// SIMATIC STEP 7 (V5.x) project Platform_V1_5
// CPU: CPU 312IFM
// CPU: CPU 313
// station: Hardware
// station: Slave
// station: P_ADR_BUS
// station: P_ADR_BUS
// station: Configuration
// station: Hardware
// station: Master
// station: P_ADR_BUS
// program: S7 Program(1)
// program: S7 Program(3)

SYMBOL_TABLE
"Ingangen.Doorsturen"	FC 1	FC 1
"Watchdog"	FC 2	FC 2
"Uitgangen.Prioriteit"	FC 3	FC 3
"Start"	I 0.0	BOOL
"Stop"	I 0.1	BOOL
"Piston A in"	I 0.2	BOOL
"Piston A uit"	I 0.3	BOOL
"Piston A onder"	I 0.4	BOOL
"Piston A boven"	I 0.5	BOOL
"Piston B in"	I 0.6	BOOL
"Piston B uit"	I 0.7	BOOL
"Piston B onder"	I 124.0	BOOL
"Piston B boven"	I 124.1	BOOL
"Proxi Pos 1"	I 124.2	BOOL
"Proxi Pos 2"	I 124.3	BOOL
"Watch.Slave.Master.Go"	M 4.0	BOOL	// Van slave Naar Master
"Watch.Slave.Master.Back"	M 4.1	BOOL	// Van slave Naar master
"Watch.Master.Slave.Go"	M 4.2	BOOL
"Watch.Master.Slave.Back"	M 4.3	BOOL
"Watch.Slave.Sim.Go"	M 4.4	BOOL
"Watch.Slave.Sim.back"	M 4.5	BOOL
"Levens.Bit"	M 10.0	BOOL
"Levens.Bit.Fout"	M 10.1	BOOL
"Ingangen 0.x"	MB 0	BYTE
"Ingangen 124.x"	MB 1	BYTE
"Uitgangen 0.x"	MB 2	BYTE
"Uitgangen 124.x"	MB 3	BYTE
"Motor Rechts"	Q 0.1	BOOL
"Piston A Op-Neer"	Q 0.2	BOOL
"Piston A Uit-In"	Q 0.3	BOOL
"Piston B Op-Neer"	Q 0.4	BOOL
"Piston B Uit-In"	Q 0.5	BOOL
"Sign.Rood"	Q 0.6	BOOL
"Motor Links"	Q 124.0	BOOL
"Extend.proxi2"	T 0	TIMER
"Levens.bit.1"	T 1	TIMER
"Levens.bit.2"	T 2	TIMER
END_SYMBOL_TABLE

FUNCTION "Ingangen.Doorsturen" : VOID	// FC 1
VERSION : 0.1
BEGIN
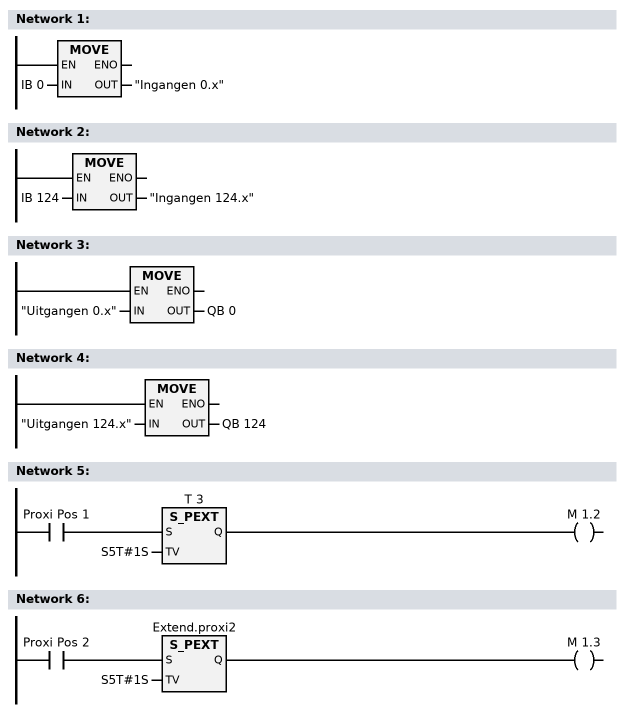
NETWORK
TITLE =
      L     IB 0;
      T     "Ingangen 0.x";
      NOP   0;
NETWORK
TITLE =
      L     IB 124;
      T     "Ingangen 124.x";
      NOP   0;
NETWORK
TITLE =
      L     "Uitgangen 0.x";
      T     QB 0;
      NOP   0;
NETWORK
TITLE =
      L     "Uitgangen 124.x";
      T     QB 124;
      NOP   0;
NETWORK
TITLE =
      A     "Proxi Pos 1";
      L     S5T#1S;
      SE    T 3;
      NOP   0;
      NOP   0;
      NOP   0;
      A     T 3;
      =     M 1.2;
NETWORK
TITLE =
      A     "Proxi Pos 2";
      L     S5T#1S;
      SE    "Extend.proxi2";
      NOP   0;
      NOP   0;
      NOP   0;
      A     "Extend.proxi2";
      =     M 1.3;
END_FUNCTION

FUNCTION "Watchdog" : VOID	// FC 2
VERSION : 0.1
BEGIN
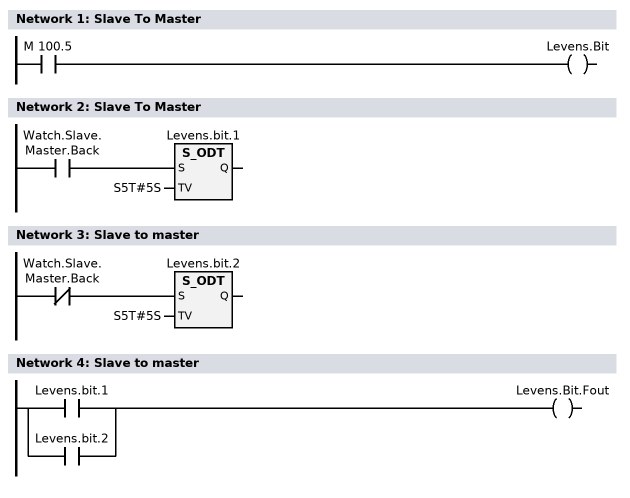
NETWORK
TITLE = Slave To Master
      A     M 100.5;
      =     "Levens.Bit";
NETWORK
TITLE = Slave To Master
      A     "Watch.Slave.Master.Back";
      L     S5T#5S;
      SD    "Levens.bit.1";
      NOP   0;
      NOP   0;
      NOP   0;
      NOP   0;
NETWORK
TITLE = Slave to master
      AN    "Watch.Slave.Master.Back";
      L     S5T#5S;
      SD    "Levens.bit.2";
      NOP   0;
      NOP   0;
      NOP   0;
      NOP   0;
NETWORK
TITLE = Slave to master
      O     "Levens.bit.1";
      O     "Levens.bit.2";
      =     "Levens.Bit.Fout";
END_FUNCTION

FUNCTION "Uitgangen.Prioriteit" : VOID	// FC 3
VERSION : 0.1
BEGIN
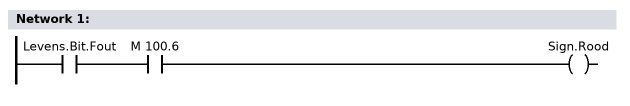
NETWORK
TITLE =
      A     "Levens.Bit.Fout";
      A     M 100.6;
      =     "Sign.Rood";
END_FUNCTION

ORGANIZATION_BLOCK OB 1
TITLE = "Main Program Sweep (Cycle)"
VERSION : 0.1
VAR_TEMP
  OB1_EV_CLASS : BYTE ;	//Bits 0-3 = 1 (Coming event), Bits 4-7 = 1 (Event class 1)
  OB1_SCAN_1 : BYTE ;	//1 (Cold restart scan 1 of OB 1), 3 (Scan 2-n of OB 1)
  OB1_PRIORITY : BYTE ;	//Priority of OB Execution
  OB1_OB_NUMBR : BYTE ;	//1 (Organization block 1, OB1)
  OB1_RESERVED_1 : BYTE ;	//Reserved for system
  OB1_RESERVED_2 : BYTE ;	//Reserved for system
  OB1_PREV_CYCLE : INT ;	//Cycle time of previous OB1 scan (milliseconds)
  OB1_MIN_CYCLE : INT ;	//Minimum cycle time of OB1 (milliseconds)
  OB1_MAX_CYCLE : INT ;	//Maximum cycle time of OB1 (milliseconds)
  OB1_DATE_TIME : DATE_AND_TIME ;	//Date and time OB1 started
END_VAR
BEGIN
NETWORK
TITLE =
      CALL  "Ingangen.Doorsturen";
      CALL  "Watchdog";
      CALL  "Uitgangen.Prioriteit";
END_ORGANIZATION_BLOCK

// (several symbol tables fit these blocks; global names not applied)

FUNCTION FC 1 : VOID
VERSION : 0.1
BEGIN
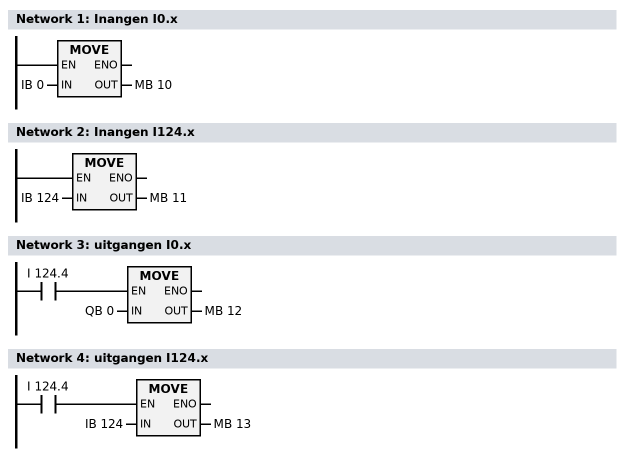
NETWORK
TITLE = Inangen I0.x
      L     IB 0;
      T     MB 10;
      NOP   0;
NETWORK
TITLE = Inangen I124.x
      L     IB 124;
      T     MB 11;
      NOP   0;
NETWORK
TITLE = uitgangen I0.x
      A     I 124.4;
      JNB   _001;
      L     QB 0;
      T     MB 12;
_001: NOP   0;
NETWORK
TITLE = uitgangen I124.x
      A     I 124.4;
      JNB   _002;
      L     IB 124;
      T     MB 13;
_002: NOP   0;
END_FUNCTION

ORGANIZATION_BLOCK OB 1
TITLE = "Main Program Sweep (Cycle)"
VERSION : 0.1
VAR_TEMP
  OB1_EV_CLASS : BYTE ;	//Bits 0-3 = 1 (Coming event), Bits 4-7 = 1 (Event class 1)
  OB1_SCAN_1 : BYTE ;	//1 (Cold restart scan 1 of OB 1), 3 (Scan 2-n of OB 1)
  OB1_PRIORITY : BYTE ;	//Priority of OB Execution
  OB1_OB_NUMBR : BYTE ;	//1 (Organization block 1, OB1)
  OB1_RESERVED_1 : BYTE ;	//Reserved for system
  OB1_RESERVED_2 : BYTE ;	//Reserved for system
  OB1_PREV_CYCLE : INT ;	//Cycle time of previous OB1 scan (milliseconds)
  OB1_MIN_CYCLE : INT ;	//Minimum cycle time of OB1 (milliseconds)
  OB1_MAX_CYCLE : INT ;	//Maximum cycle time of OB1 (milliseconds)
  OB1_DATE_TIME : DATE_AND_TIME ;	//Date and time OB1 started
END_VAR
BEGIN
// (block stored without names or comments; labels and parameter names are numbered)
END_ORGANIZATION_BLOCK

SYMBOL_TABLE
"Productie_teller_Station"	C 0	COUNTER
"Productie_teller_Stat_A"	C 1	COUNTER
"Productie_teller_Stat_B"	C 2	COUNTER
"Productie_teller_In_Waar"	C 3	COUNTER
"SIM.Positie.Staven"	C 4	COUNTER
"SIM.OB1"	DB 2	DB 2	// Simualtie
"SIM.USERS"	DB 3	DB 3
"Positionering"	DB 4	DB 4
"Uitgangen Sturen"	FC 1	FC 1
"Timers + Counters"	FC 2	FC 2
"Grafcet Station A"	FC 3	FC 3
"Grafcet Station B"	FC 4	FC 4
"Simulatie_Run"	FC 5	FC 5
"Opstart_FC"	FC 6	FC 6
"Grafcet_Platform"	FC 7	FC 7	// Grafcet_Platform
"Ingang -> Merker"	FC 8	FC 8
"DB_Function"	FC 9	FC 9
"SIM.OB100"	FC 10	FC 10
"SIM.user"	FC 11	FC 11
"Positionering_balken"	FC 12	FC 12
"Sub_routine"	FC 14	FC 14
"Opstart_subroutine"	FC 15	FC 15
"Sub_routine_gelijk"	FC 16	FC 16
"Sub_route_Station_samen"	FC 17	FC 17
"SIM.SUBR.Y-As"	FC 19	FC 19
"SIM.LOGIN"	FC 20	FC 20
"SIM.Move.X-As"	FC 21	FC 21
"SIM.BALK.Reset"	FC 22	FC 22
"Stap 0.0"	M 0.0	BOOL
"Stap 0.1"	M 0.1	BOOL
"Stap 0.2"	M 0.2	BOOL
"Stap 0.3"	M 0.3	BOOL
"Stap 0.4"	M 0.4	BOOL
"Stap 0.5"	M 0.5	BOOL
"Stap 1.1"	M 1.1	BOOL
"Stap 1.2"	M 1.2	BOOL
"Stap 1.3"	M 1.3	BOOL
"Stap 1.4"	M 1.4	BOOL
"Stap 1.5"	M 1.5	BOOL
"Stap 2.0"	M 2.0	BOOL
"Stap 2.1"	M 2.1	BOOL
"Stap 2.2"	M 2.2	BOOL
"Stap 2.3"	M 2.3	BOOL
"Stap 2.4"	M 2.4	BOOL
"Stap 2.5"	M 2.5	BOOL
"Start"	M 5.0	BOOL
"Stop"	M 5.1	BOOL
"Piston A in"	M 5.2	BOOL
"Piston A uit"	M 5.3	BOOL
"Piston A onder"	M 5.4	BOOL
"Piston A boven"	M 5.5	BOOL
"Piston B in"	M 5.6	BOOL
"Piston B uit"	M 5.7	BOOL
"Piston B onder"	M 6.0	BOOL
"Piston B boven"	M 6.1	BOOL
"Proxi Pos 1"	M 6.2	BOOL
"Proxi Pos 2"	M 6.3	BOOL
"Motor Rechts"	M 7.1	BOOL
"Piston A Op-Neer"	M 7.2	BOOL
"Piston A Uit-In"	M 7.3	BOOL
"Piston B Op-Neer"	M 7.4	BOOL
"Piston B Uit-In"	M 7.5	BOOL
"Sign.Rood"	M 7.6	BOOL
"Sign.Groen"	M 7.7	BOOL
"Motor Links"	M 8.0	BOOL
"Opstart"	M 10.0	BOOL
"SIM.reset.C4"	M 10.1	BOOL
"P.M10.2"	M 10.2	BOOL
"SIM.opstart.5S"	M 10.3	BOOL
"admin"	M 11.0	BOOL
"monitor"	M 11.1	BOOL
"operate"	M 11.2	BOOL
"user"	M 11.3	BOOL
"SIM.User.Login"	M 11.4	BOOL
"SIM.User.logout"	M 11.5	BOOL
"SIM.USER.ERROR"	M 11.6	BOOL
"Sim.Start.Postitionering"	M 24.0	BOOL
"Postitionering.Station.A"	M 24.1	BOOL
"Postitionering.Station.B"	M 24.2	BOOL
"Postitionering.Return"	M 24.3	BOOL
"SIM.Positie.Save"	M 24.4	BOOL
"SIM.Positie.Zoom"	M 24.5	BOOL
"Balk1"	M 25.0	BOOL
"Blak2"	M 25.1	BOOL
"Balk3"	M 25.2	BOOL
"Balk4"	M 25.3	BOOL
"Balk5"	M 25.4	BOOL
"Balk6"	M 25.5	BOOL
"Balk7"	M 25.6	BOOL
"Balk8"	M 25.7	BOOL
"Test Piston A"	M 30.0	BOOL
"Fout Controle station A"	M 30.1	BOOL
"Fout Reset station A"	M 30.2	BOOL
"Test station B"	M 30.3	BOOL
"Fout Controle station B"	M 30.4	BOOL
"Fout_Motor"	M 30.5	BOOL
"Foint Station_A_B"	M 30.6	BOOL
"Stop Meker"	M 30.7	BOOL
"DBW0 == DBW2"	M 31.0	BOOL
"DBW0 < DBW2"	M 31.1	BOOL
"DBW0 != 0"	M 31.2	BOOL
"SIM.Start.StaA"	M 31.3	BOOL
"SIM.Start.StaB"	M 31.4	BOOL
"SIM.Start"	M 31.5	BOOL
"SIM.Stop"	M 31.6	BOOL
"DBW0 == 0"	M 32.0	BOOL
"INI.Stations"	M 33.0	BOOL
"Start Stat A + B"	M 33.1	BOOL
"Blinker 5s"	M 100.5	BOOL
"Restart"	M 101.1	BOOL
"Ingangen 0.x"	MB 5	BYTE
"Ingangen 124.x"	MB 6	BYTE
"Uitgangen 0.x"	MB 7	BYTE
"Uitgangen 124.x"	MB 8	BYTE
"Positie.balken"	MB 25	BYTE
"SIM.C.Positie.BCD"	MW 12	WORD	// Balk die zich bevind voor de sensoren(bcd waarde)
"SIM.C.Positie.INT"	MW 14	INT	// Balk die zich bevind voor de sensoren(int waarde)
"SIM.C.Postie.Stat.A"	MW 16	INT	// Balk die zich bevind voor station A
"SIM.C.Postie.Stat.B"	MW 18	INT	// Balk due zich bevind voor station B
"SIM.Station.A"	MW 20	WORD
"SIM.Station.B"	MW 22	WORD
"COMPLETE RESTART"	OB 100	OB 100	// Complete Restart
"Motor controler"	T 0	TIMER
"Timer Contr Neer A"	T 1	TIMER
"Timer contr uit A"	T 2	TIMER
"Timer contr uit B"	T 3	TIMER
"Timer contr neer B"	T 4	TIMER
"Hori Station B"	T 5	TIMER
"Verti Station B"	T 6	TIMER
"SIM.SUBR.T1"	T 7	TIMER
"SIM.SUBR.T2"	T 8	TIMER
"SIM.User.Error.T"	T 9	TIMER
"Vertraging.Station.off"	T 10	TIMER
"Vertraging.Station.Aan"	T 11	TIMER
END_SYMBOL_TABLE

FUNCTION "Uitgangen Sturen" : VOID	// FC 1
VERSION : 0.1
BEGIN
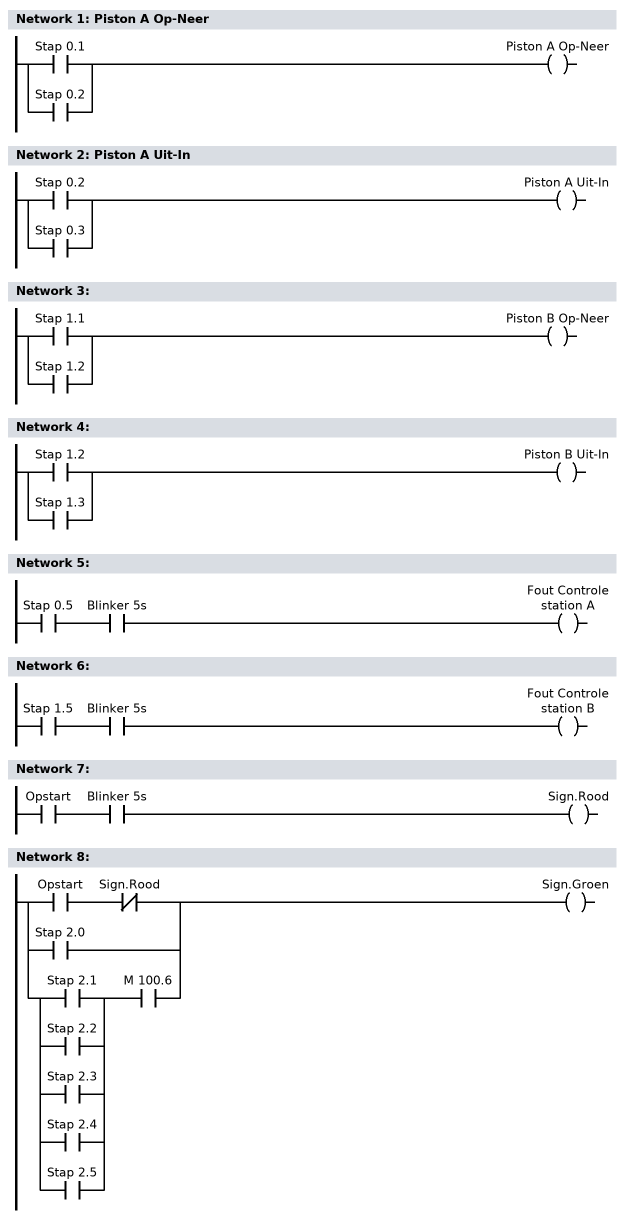
NETWORK
TITLE = Piston A Op-Neer
      O     "Stap 0.1";
      O     "Stap 0.2";
      =     "Piston A Op-Neer";
NETWORK
TITLE = Piston A Uit-In
      O     "Stap 0.2";
      O     "Stap 0.3";
      =     "Piston A Uit-In";
NETWORK
TITLE =
      O     "Stap 1.1";
      O     "Stap 1.2";
      =     "Piston B Op-Neer";
NETWORK
TITLE =
      O     "Stap 1.2";
      O     "Stap 1.3";
      =     "Piston B Uit-In";
NETWORK
TITLE =
      A     "Stap 0.5";
      A     "Blinker 5s";
      =     "Fout Controle station A";
NETWORK
TITLE =
      A     "Stap 1.5";
      A     "Blinker 5s";
      =     "Fout Controle station B";
NETWORK
TITLE =
      A     "Opstart";
      A     "Blinker 5s";
      =     "Sign.Rood";
NETWORK
TITLE =
      A     "Opstart";
      AN    "Sign.Rood";
      O     "Stap 2.0";
      O;
      A(;
      O     "Stap 2.1";
      O     "Stap 2.2";
      O     "Stap 2.3";
      O     "Stap 2.4";
      O     "Stap 2.5";
      );
      A     M 100.6;
      =     "Sign.Groen";
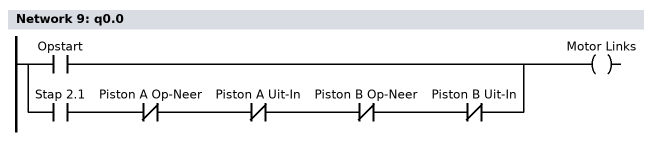
NETWORK
TITLE = q0.0
      O     "Opstart";
      O;
      A     "Stap 2.1";
      AN    "Piston A Op-Neer";
      AN    "Piston A Uit-In";
      AN    "Piston B Op-Neer";
      AN    "Piston B Uit-In";
      =     "Motor Links";
END_FUNCTION

FUNCTION "Timers + Counters" : VOID	// FC 2
VERSION : 0.1
BEGIN
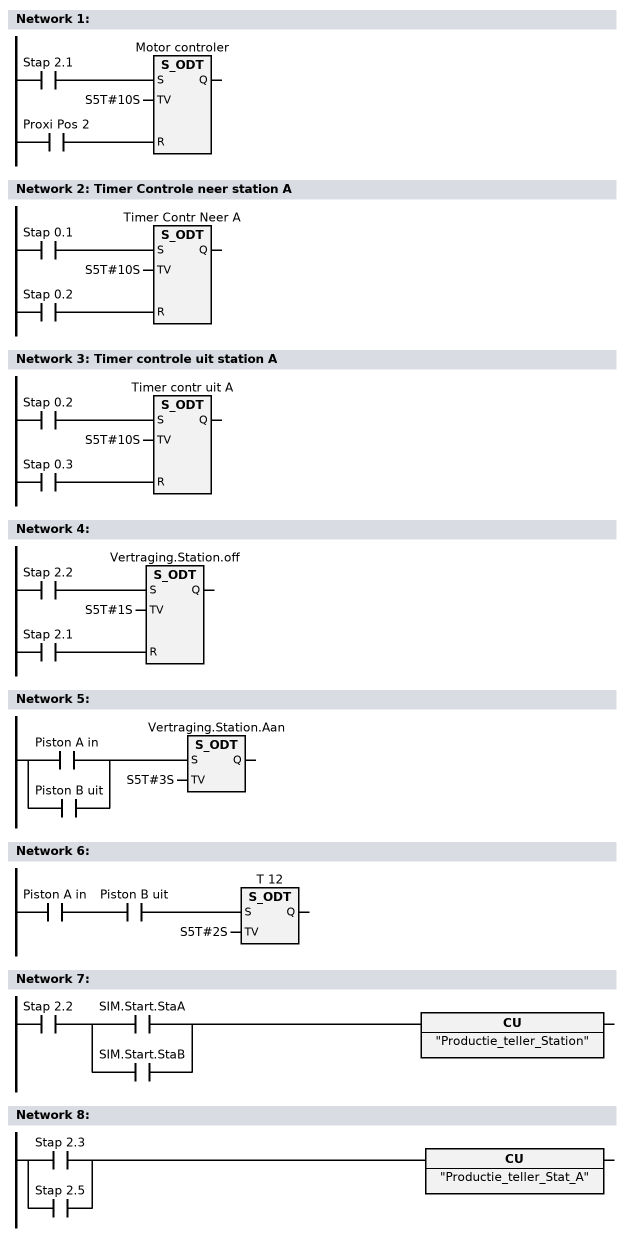
NETWORK
TITLE =
      A     "Stap 2.1";
      L     S5T#10S;
      SD    "Motor controler";
      A     "Proxi Pos 2";
      R     "Motor controler";
      NOP   0;
      NOP   0;
      NOP   0;
NETWORK
TITLE = Timer Controle neer station A
      A     "Stap 0.1";
      L     S5T#10S;
      SD    "Timer Contr Neer A";
      A     "Stap 0.2";
      R     "Timer Contr Neer A";
      NOP   0;
      NOP   0;
      NOP   0;
NETWORK
TITLE = Timer controle uit station A
      A     "Stap 0.2";
      L     S5T#10S;
      SD    "Timer contr uit A";
      A     "Stap 0.3";
      R     "Timer contr uit A";
      NOP   0;
      NOP   0;
      NOP   0;
NETWORK
TITLE =
      A     "Stap 2.2";
      L     S5T#1S;
      SD    "Vertraging.Station.off";
      A     "Stap 2.1";
      R     "Vertraging.Station.off";
      NOP   0;
      NOP   0;
      NOP   0;
NETWORK
TITLE =
      A(;
      O     "Piston A in";
      O     "Piston B uit";
      );
      L     S5T#3S;
      SD    "Vertraging.Station.Aan";
      NOP   0;
      NOP   0;
      NOP   0;
      NOP   0;
NETWORK
TITLE =
      A     "Piston A in";
      A     "Piston B uit";
      L     S5T#2S;
      SD    T 12;
      NOP   0;
      NOP   0;
      NOP   0;
      NOP   0;
NETWORK
TITLE =
      A     "Stap 2.2";
      A(;
      O     "SIM.Start.StaA";
      O     "SIM.Start.StaB";
      );
      CU    "Productie_teller_Station";
      BLD   101;
      NOP   0;
      NOP   0;
      NOP   0;
      NOP   0;
      NOP   0;
      NOP   0;
NETWORK
TITLE =
      A(;
      O     "Stap 2.3";
      O     "Stap 2.5";
      );
      CU    "Productie_teller_Stat_A";
      BLD   101;
      NOP   0;
      NOP   0;
      NOP   0;
      NOP   0;
      NOP   0;
      NOP   0;
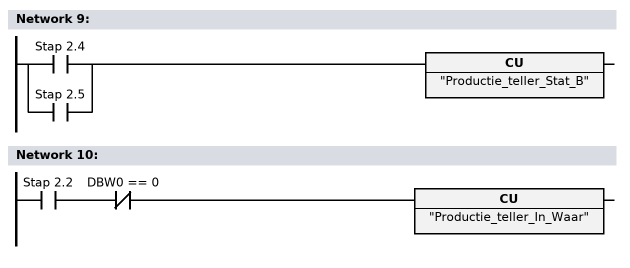
NETWORK
TITLE =
      A(;
      O     "Stap 2.4";
      O     "Stap 2.5";
      );
      CU    "Productie_teller_Stat_B";
      BLD   101;
      NOP   0;
      NOP   0;
      NOP   0;
      NOP   0;
      NOP   0;
      NOP   0;
NETWORK
TITLE =
      A     "Stap 2.2";
      AN    "DBW0 == 0";
      CU    "Productie_teller_In_Waar";
      BLD   101;
      NOP   0;
      NOP   0;
      NOP   0;
      NOP   0;
      NOP   0;
      NOP   0;
END_FUNCTION

FUNCTION "Grafcet Station A" : VOID	// FC 3
VERSION : 0.1
BEGIN
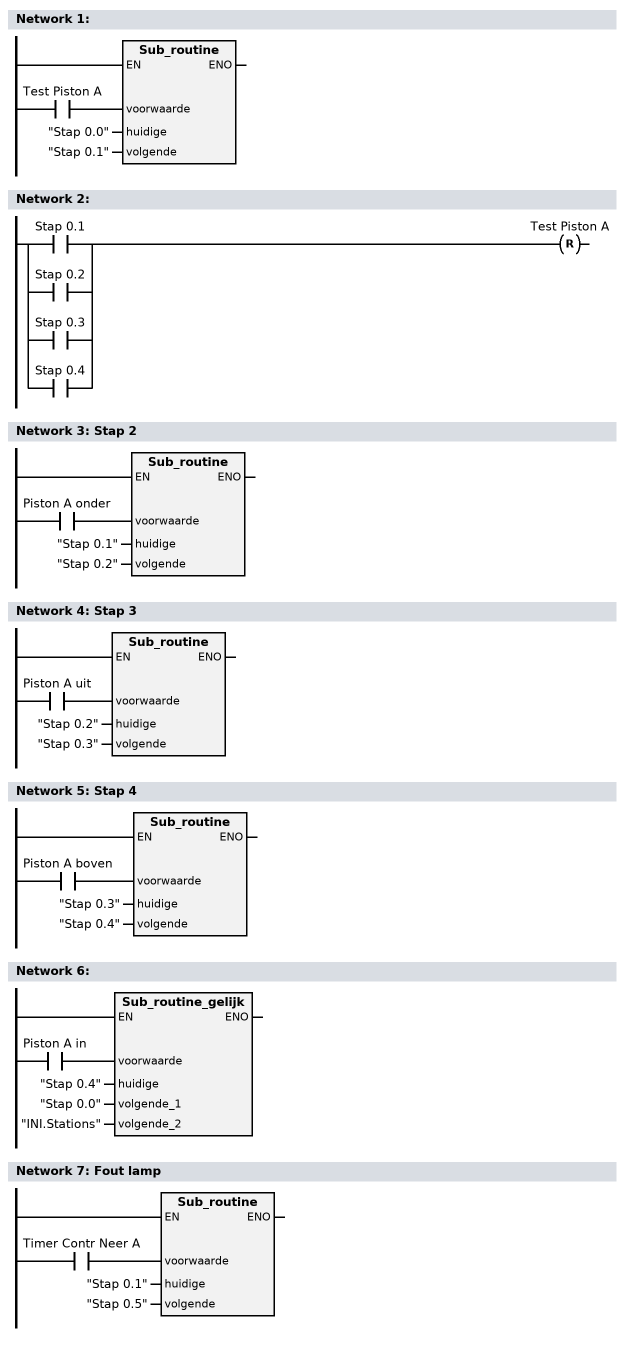
NETWORK
TITLE =
      A     "Test Piston A";
      =     L 0.0;
      BLD   103;
      CALL  "Sub_routine" (
           voorwaarde               := L 0.0,
           huidige                  := "Stap 0.0",
           volgende                 := "Stap 0.1");
      NOP   0;
NETWORK
TITLE =
      O     "Stap 0.1";
      O     "Stap 0.2";
      O     "Stap 0.3";
      O     "Stap 0.4";
      R     "Test Piston A";
NETWORK
TITLE = Stap 2
      A     "Piston A onder";
      =     L 0.0;
      BLD   103;
      CALL  "Sub_routine" (
           voorwaarde               := L 0.0,
           huidige                  := "Stap 0.1",
           volgende                 := "Stap 0.2");
      NOP   0;
NETWORK
TITLE = Stap 3
      A     "Piston A uit";
      =     L 0.0;
      BLD   103;
      CALL  "Sub_routine" (
           voorwaarde               := L 0.0,
           huidige                  := "Stap 0.2",
           volgende                 := "Stap 0.3");
      NOP   0;
NETWORK
TITLE = Stap 4
      A     "Piston A boven";
      =     L 0.0;
      BLD   103;
      CALL  "Sub_routine" (
           voorwaarde               := L 0.0,
           huidige                  := "Stap 0.3",
           volgende                 := "Stap 0.4");
      NOP   0;
NETWORK
TITLE =
      A     "Piston A in";
      =     L 0.0;
      BLD   103;
      CALL  "Sub_routine_gelijk" (
           voorwaarde               := L 0.0,
           huidige                  := "Stap 0.4",
           volgende_1               := "Stap 0.0",
           volgende_2               := "INI.Stations");
      NOP   0;
NETWORK
TITLE = Fout lamp
      A     "Timer Contr Neer A";
      =     L 0.0;
      BLD   103;
      CALL  "Sub_routine" (
           voorwaarde               := L 0.0,
           huidige                  := "Stap 0.1",
           volgende                 := "Stap 0.5");
      NOP   0;
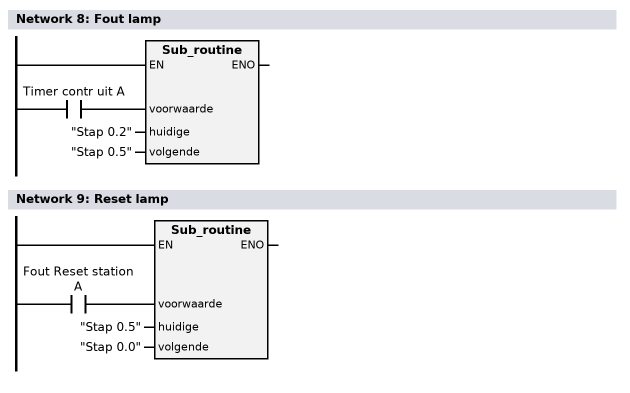
NETWORK
TITLE = Fout lamp
      A     "Timer contr uit A";
      =     L 0.0;
      BLD   103;
      CALL  "Sub_routine" (
           voorwaarde               := L 0.0,
           huidige                  := "Stap 0.2",
           volgende                 := "Stap 0.5");
      NOP   0;
NETWORK
TITLE = Reset lamp
      A     "Fout Reset station A";
      =     L 0.0;
      BLD   103;
      CALL  "Sub_routine" (
           voorwaarde               := L 0.0,
           huidige                  := "Stap 0.5",
           volgende                 := "Stap 0.0");
      NOP   0;
END_FUNCTION

FUNCTION "Grafcet Station B" : VOID	// FC 4
VERSION : 0.1
BEGIN
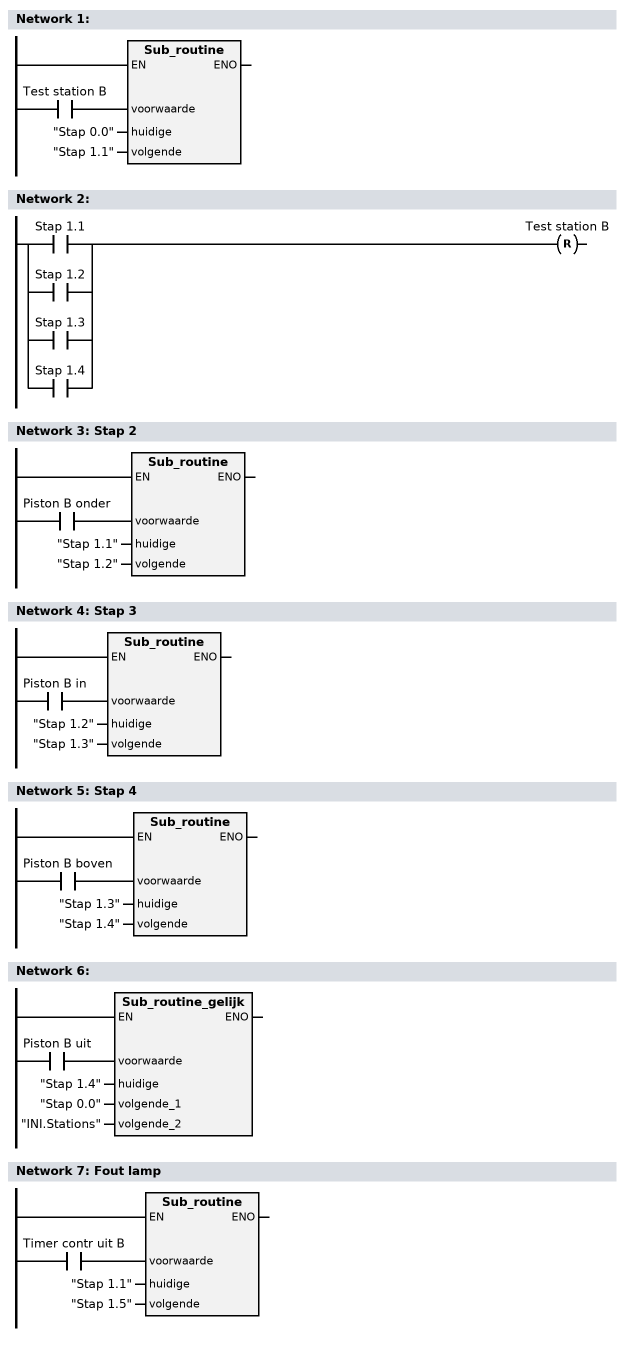
NETWORK
TITLE =
      A     "Test station B";
      =     L 0.0;
      BLD   103;
      CALL  "Sub_routine" (
           voorwaarde               := L 0.0,
           huidige                  := "Stap 0.0",
           volgende                 := "Stap 1.1");
      NOP   0;
NETWORK
TITLE =
      O     "Stap 1.1";
      O     "Stap 1.2";
      O     "Stap 1.3";
      O     "Stap 1.4";
      R     "Test station B";
NETWORK
TITLE = Stap 2
      A     "Piston B onder";
      =     L 0.0;
      BLD   103;
      CALL  "Sub_routine" (
           voorwaarde               := L 0.0,
           huidige                  := "Stap 1.1",
           volgende                 := "Stap 1.2");
      NOP   0;
NETWORK
TITLE = Stap 3
      A     "Piston B in";
      =     L 0.0;
      BLD   103;
      CALL  "Sub_routine" (
           voorwaarde               := L 0.0,
           huidige                  := "Stap 1.2",
           volgende                 := "Stap 1.3");
      NOP   0;
NETWORK
TITLE = Stap 4
      A     "Piston B boven";
      =     L 0.0;
      BLD   103;
      CALL  "Sub_routine" (
           voorwaarde               := L 0.0,
           huidige                  := "Stap 1.3",
           volgende                 := "Stap 1.4");
      NOP   0;
NETWORK
TITLE =
      A     "Piston B uit";
      =     L 0.0;
      BLD   103;
      CALL  "Sub_routine_gelijk" (
           voorwaarde               := L 0.0,
           huidige                  := "Stap 1.4",
           volgende_1               := "Stap 0.0",
           volgende_2               := "INI.Stations");
      NOP   0;
NETWORK
TITLE = Fout lamp
      A     "Timer contr uit B";
      =     L 0.0;
      BLD   103;
      CALL  "Sub_routine" (
           voorwaarde               := L 0.0,
           huidige                  := "Stap 1.1",
           volgende                 := "Stap 1.5");
      NOP   0;
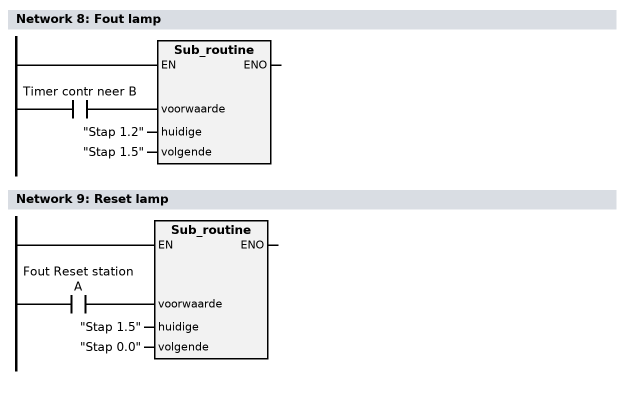
NETWORK
TITLE = Fout lamp
      A     "Timer contr neer B";
      =     L 0.0;
      BLD   103;
      CALL  "Sub_routine" (
           voorwaarde               := L 0.0,
           huidige                  := "Stap 1.2",
           volgende                 := "Stap 1.5");
      NOP   0;
NETWORK
TITLE = Reset lamp
      A     "Fout Reset station A";
      =     L 0.0;
      BLD   103;
      CALL  "Sub_routine" (
           voorwaarde               := L 0.0,
           huidige                  := "Stap 1.5",
           volgende                 := "Stap 0.0");
      NOP   0;
END_FUNCTION

FUNCTION "Simulatie_Run" : VOID	// FC 5
VERSION : 0.1
BEGIN
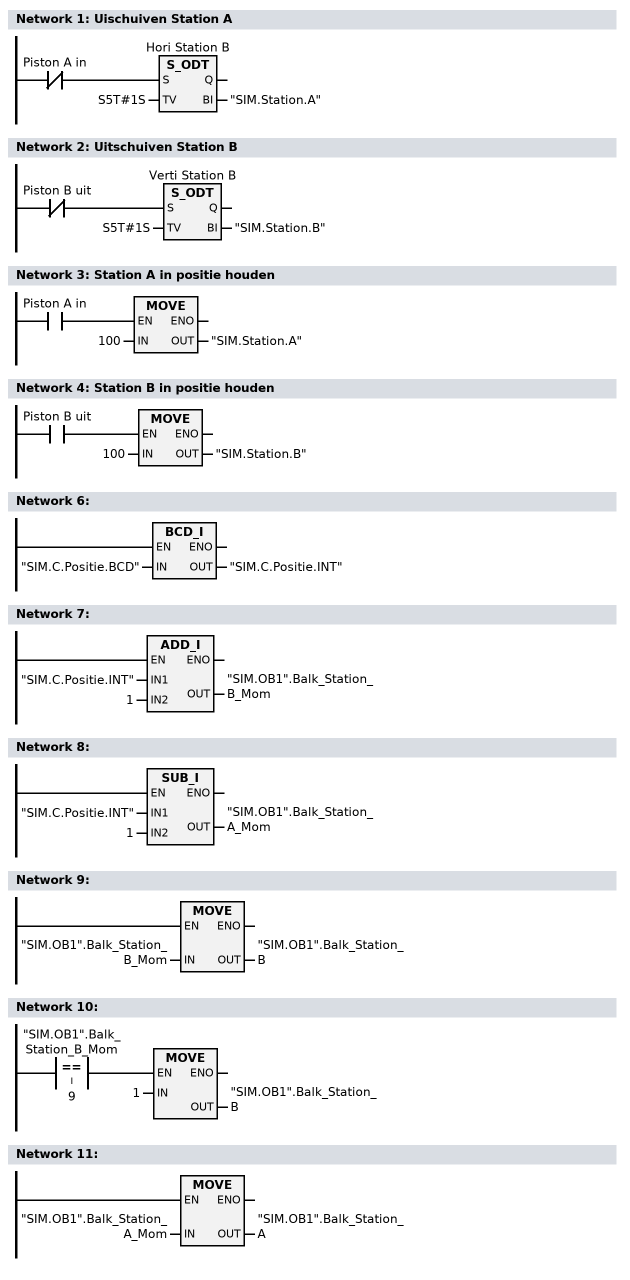
NETWORK
TITLE = Uischuiven Station A
      AN    "Piston A in";
      L     S5T#1S;
      SD    "Hori Station B";
      NOP   0;
      L     "Hori Station B";
      T     "SIM.Station.A";
      NOP   0;
      NOP   0;
NETWORK
TITLE = Uitschuiven Station B
      AN    "Piston B uit";
      L     S5T#1S;
      SD    "Verti Station B";
      NOP   0;
      L     "Verti Station B";
      T     "SIM.Station.B";
      NOP   0;
      NOP   0;
NETWORK
TITLE = Station A in positie houden
      A     "Piston A in";
      JNB   _001;
      L     100;
      T     "SIM.Station.A";
_001: NOP   0;
NETWORK
TITLE = Station B in positie houden
      A     "Piston B uit";
      JNB   _002;
      L     100;
      T     "SIM.Station.B";
_002: NOP   0;
NETWORK
TITLE = Balk voor de sensoren
      A     "Proxi Pos 2";
      AN    "Proxi Pos 1";
      FP    M 40.0;
      CU    "SIM.Positie.Staven";
      BLD   101;
      A     "Proxi Pos 1";
      FP    M 40.1;
      L     C#1;
      S     "SIM.Positie.Staven";
      NOP   0;
      NOP   0;
      LC    "SIM.Positie.Staven";
      T     "SIM.C.Positie.BCD";
      NOP   0;
NETWORK
TITLE =
      L     "SIM.C.Positie.BCD";
      BTI;
      T     "SIM.C.Positie.INT";
      NOP   0;
NETWORK
TITLE =
      L     "SIM.C.Positie.INT";
      L     1;
      +I;
      T     "SIM.OB1".Balk_Station_B_Mom;
      NOP   0;
NETWORK
TITLE =
      L     "SIM.C.Positie.INT";
      L     1;
      -I;
      T     "SIM.OB1".Balk_Station_A_Mom;
      NOP   0;
NETWORK
TITLE =
      L     "SIM.OB1".Balk_Station_B_Mom;
      T     "SIM.OB1".Balk_Station_B;
      NOP   0;
NETWORK
TITLE =
      A(;
      L     "SIM.OB1".Balk_Station_B_Mom;
      L     9;
      ==I;
      );
      JNB   _003;
      L     1;
      T     "SIM.OB1".Balk_Station_B;
_003: NOP   0;
NETWORK
TITLE =
      L     "SIM.OB1".Balk_Station_A_Mom;
      T     "SIM.OB1".Balk_Station_A;
      NOP   0;
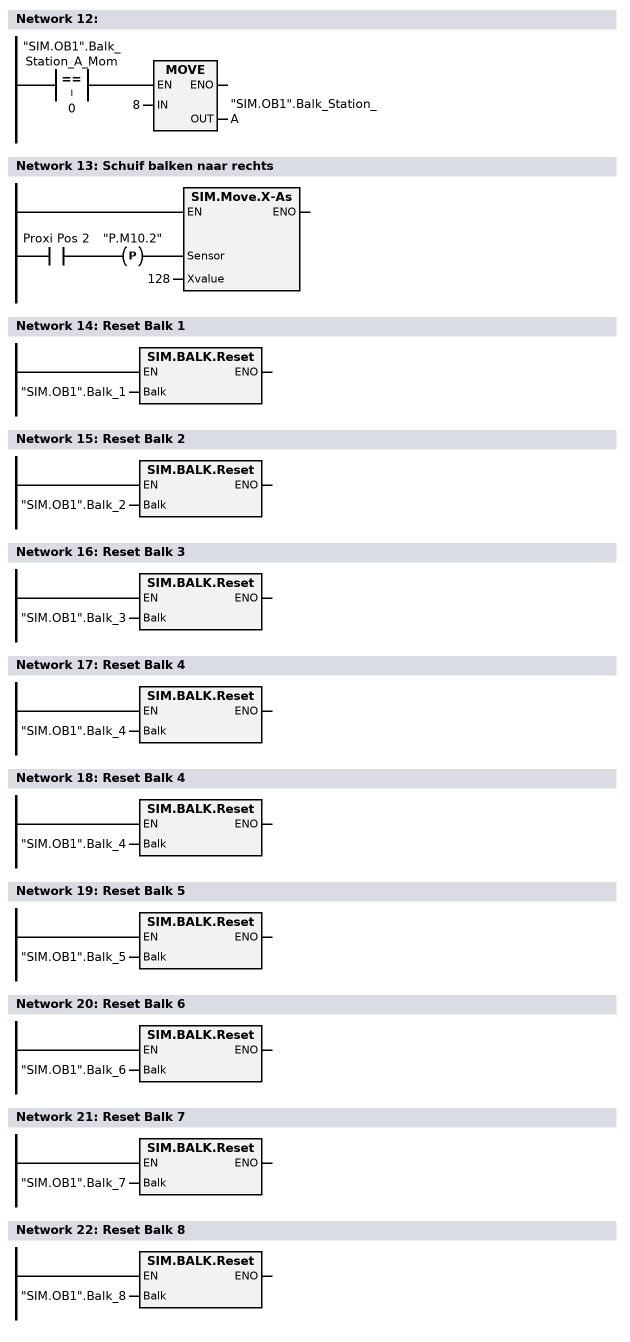
NETWORK
TITLE =
      A(;
      L     "SIM.OB1".Balk_Station_A_Mom;
      L     0;
      ==I;
      );
      JNB   _004;
      L     8;
      T     "SIM.OB1".Balk_Station_A;
_004: NOP   0;
NETWORK
TITLE = Schuif balken naar rechts
      A     "Proxi Pos 2";
      FP    "P.M10.2";
      =     L 0.0;
      BLD   103;
      CALL  "SIM.Move.X-As" (
           Sensor                   := L 0.0,
           Xvalue                   := 128);
      NOP   0;
NETWORK
TITLE = Reset Balk 1
      CALL  "SIM.BALK.Reset" (
           Balk                     := "SIM.OB1".Balk_1);
      NOP   0;
NETWORK
TITLE = Reset Balk 2
      CALL  "SIM.BALK.Reset" (
           Balk                     := "SIM.OB1".Balk_2);
      NOP   0;
NETWORK
TITLE = Reset Balk 3
      CALL  "SIM.BALK.Reset" (
           Balk                     := "SIM.OB1".Balk_3);
      NOP   0;
NETWORK
TITLE = Reset Balk 4
      CALL  "SIM.BALK.Reset" (
           Balk                     := "SIM.OB1".Balk_4);
      NOP   0;
NETWORK
TITLE = Reset Balk 4
      CALL  "SIM.BALK.Reset" (
           Balk                     := "SIM.OB1".Balk_4);
      NOP   0;
NETWORK
TITLE = Reset Balk 5
      CALL  "SIM.BALK.Reset" (
           Balk                     := "SIM.OB1".Balk_5);
      NOP   0;
NETWORK
TITLE = Reset Balk 6
      CALL  "SIM.BALK.Reset" (
           Balk                     := "SIM.OB1".Balk_6);
      NOP   0;
NETWORK
TITLE = Reset Balk 7
      CALL  "SIM.BALK.Reset" (
           Balk                     := "SIM.OB1".Balk_7);
      NOP   0;
NETWORK
TITLE = Reset Balk 8
      CALL  "SIM.BALK.Reset" (
           Balk                     := "SIM.OB1".Balk_8);
      NOP   0;
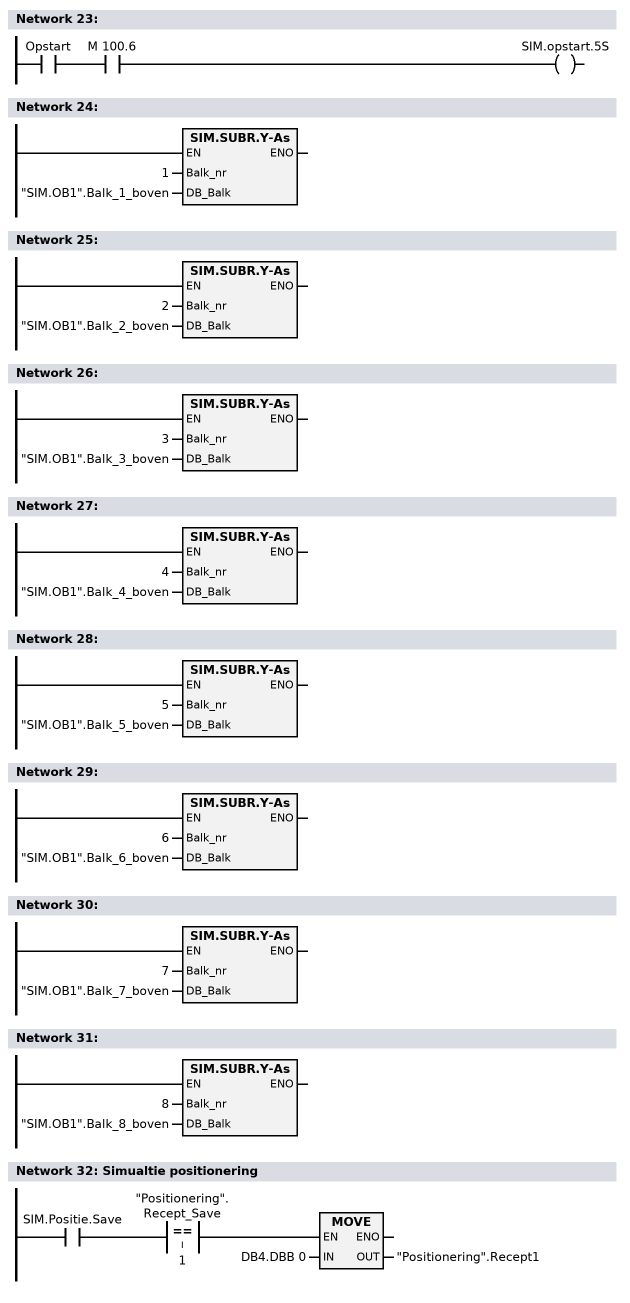
NETWORK
TITLE =
      A     "Opstart";
      A     M 100.6;
      =     "SIM.opstart.5S";
NETWORK
TITLE =
      CALL  "SIM.SUBR.Y-As" (
           Balk_nr                  := 1,
           DB_Balk                  := "SIM.OB1".Balk_1_boven);
      NOP   0;
NETWORK
TITLE =
      CALL  "SIM.SUBR.Y-As" (
           Balk_nr                  := 2,
           DB_Balk                  := "SIM.OB1".Balk_2_boven);
      NOP   0;
NETWORK
TITLE =
      CALL  "SIM.SUBR.Y-As" (
           Balk_nr                  := 3,
           DB_Balk                  := "SIM.OB1".Balk_3_boven);
      NOP   0;
NETWORK
TITLE =
      CALL  "SIM.SUBR.Y-As" (
           Balk_nr                  := 4,
           DB_Balk                  := "SIM.OB1".Balk_4_boven);
      NOP   0;
NETWORK
TITLE =
      CALL  "SIM.SUBR.Y-As" (
           Balk_nr                  := 5,
           DB_Balk                  := "SIM.OB1".Balk_5_boven);
      NOP   0;
NETWORK
TITLE =
      CALL  "SIM.SUBR.Y-As" (
           Balk_nr                  := 6,
           DB_Balk                  := "SIM.OB1".Balk_6_boven);
      NOP   0;
NETWORK
TITLE =
      CALL  "SIM.SUBR.Y-As" (
           Balk_nr                  := 7,
           DB_Balk                  := "SIM.OB1".Balk_7_boven);
      NOP   0;
NETWORK
TITLE =
      CALL  "SIM.SUBR.Y-As" (
           Balk_nr                  := 8,
           DB_Balk                  := "SIM.OB1".Balk_8_boven);
      NOP   0;
NETWORK
TITLE = Simualtie positionering
      A     "SIM.Positie.Save";
      A(;
      L     "Positionering".Recept_Save;
      L     1;
      ==I;
      );
      JNB   _005;
      L     DB4.DBB 0;
      T     "Positionering".Recept1;
_005: NOP   0;
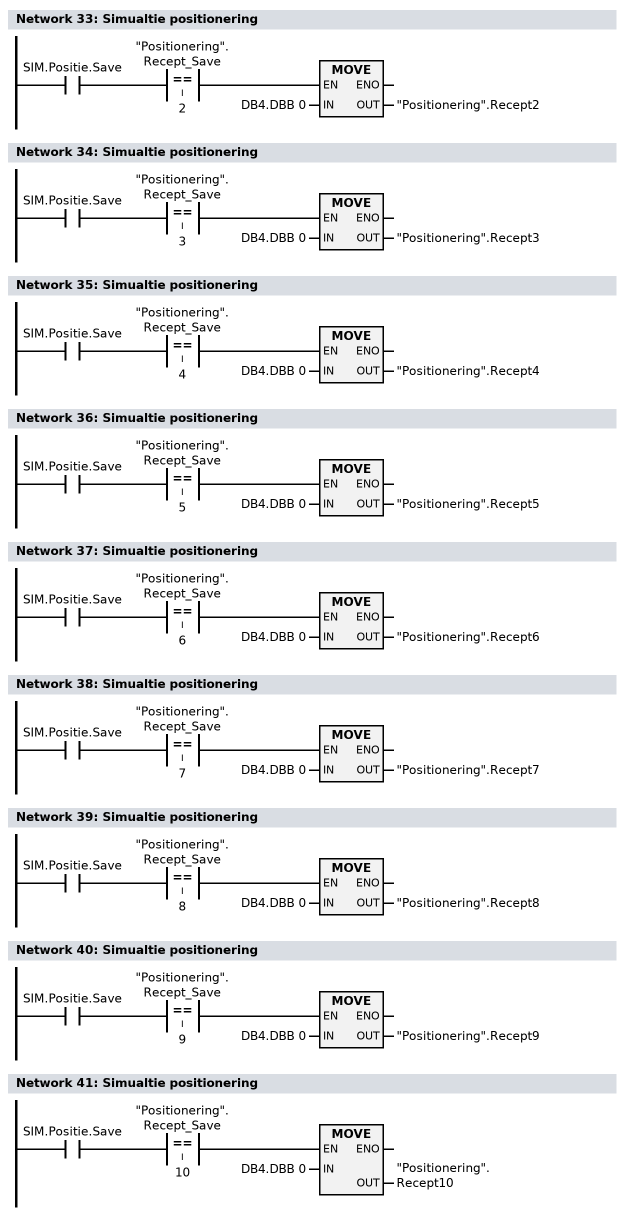
NETWORK
TITLE = Simualtie positionering
      A     "SIM.Positie.Save";
      A(;
      L     "Positionering".Recept_Save;
      L     2;
      ==I;
      );
      JNB   _006;
      L     DB4.DBB 0;
      T     "Positionering".Recept2;
_006: NOP   0;
NETWORK
TITLE = Simualtie positionering
      A     "SIM.Positie.Save";
      A(;
      L     "Positionering".Recept_Save;
      L     3;
      ==I;
      );
      JNB   _007;
      L     DB4.DBB 0;
      T     "Positionering".Recept3;
_007: NOP   0;
NETWORK
TITLE = Simualtie positionering
      A     "SIM.Positie.Save";
      A(;
      L     "Positionering".Recept_Save;
      L     4;
      ==I;
      );
      JNB   _008;
      L     DB4.DBB 0;
      T     "Positionering".Recept4;
_008: NOP   0;
NETWORK
TITLE = Simualtie positionering
      A     "SIM.Positie.Save";
      A(;
      L     "Positionering".Recept_Save;
      L     5;
      ==I;
      );
      JNB   _009;
      L     DB4.DBB 0;
      T     "Positionering".Recept5;
_009: NOP   0;
NETWORK
TITLE = Simualtie positionering
      A     "SIM.Positie.Save";
      A(;
      L     "Positionering".Recept_Save;
      L     6;
      ==I;
      );
      JNB   _00a;
      L     DB4.DBB 0;
      T     "Positionering".Recept6;
_00a: NOP   0;
NETWORK
TITLE = Simualtie positionering
      A     "SIM.Positie.Save";
      A(;
      L     "Positionering".Recept_Save;
      L     7;
      ==I;
      );
      JNB   _00b;
      L     DB4.DBB 0;
      T     "Positionering".Recept7;
_00b: NOP   0;
NETWORK
TITLE = Simualtie positionering
      A     "SIM.Positie.Save";
      A(;
      L     "Positionering".Recept_Save;
      L     8;
      ==I;
      );
      JNB   _00c;
      L     DB4.DBB 0;
      T     "Positionering".Recept8;
_00c: NOP   0;
NETWORK
TITLE = Simualtie positionering
      A     "SIM.Positie.Save";
      A(;
      L     "Positionering".Recept_Save;
      L     9;
      ==I;
      );
      JNB   _00d;
      L     DB4.DBB 0;
      T     "Positionering".Recept9;
_00d: NOP   0;
NETWORK
TITLE = Simualtie positionering
      A     "SIM.Positie.Save";
      A(;
      L     "Positionering".Recept_Save;
      L     10;
      ==I;
      );
      JNB   _00e;
      L     DB4.DBB 0;
      T     "Positionering".Recept10;
_00e: NOP   0;
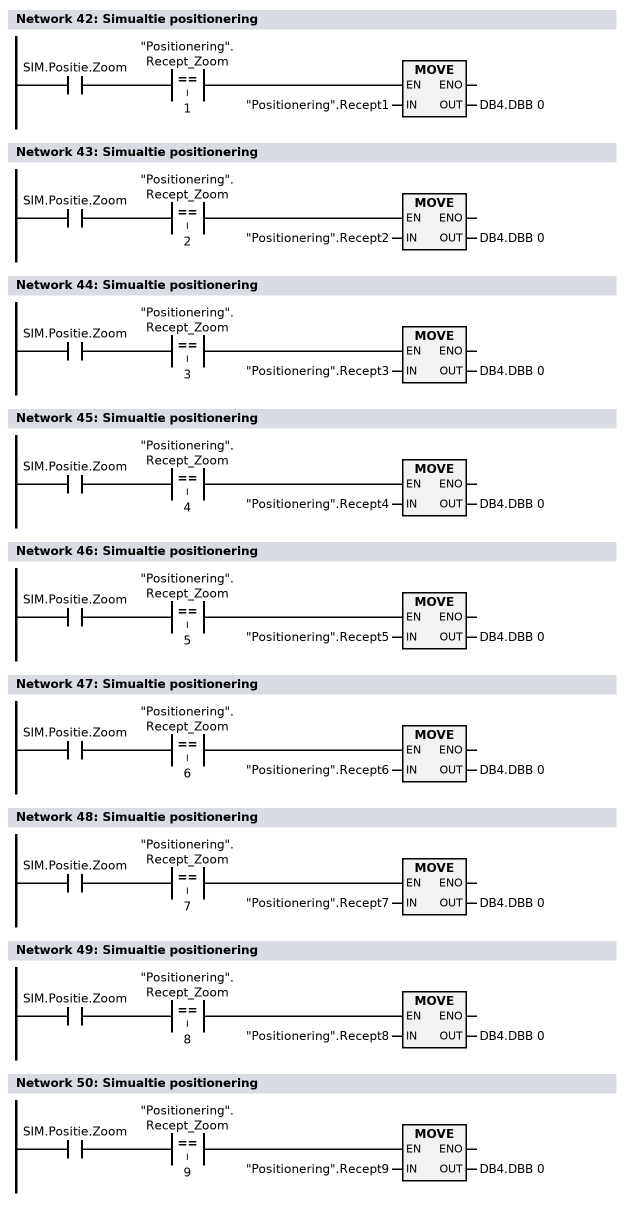
NETWORK
TITLE = Simualtie positionering
      A     "SIM.Positie.Zoom";
      A(;
      L     "Positionering".Recept_Zoom;
      L     1;
      ==I;
      );
      JNB   _00f;
      L     "Positionering".Recept1;
      T     DB4.DBB 0;
_00f: NOP   0;
NETWORK
TITLE = Simualtie positionering
      A     "SIM.Positie.Zoom";
      A(;
      L     "Positionering".Recept_Zoom;
      L     2;
      ==I;
      );
      JNB   _010;
      L     "Positionering".Recept2;
      T     DB4.DBB 0;
_010: NOP   0;
NETWORK
TITLE = Simualtie positionering
      A     "SIM.Positie.Zoom";
      A(;
      L     "Positionering".Recept_Zoom;
      L     3;
      ==I;
      );
      JNB   _011;
      L     "Positionering".Recept3;
      T     DB4.DBB 0;
_011: NOP   0;
NETWORK
TITLE = Simualtie positionering
      A     "SIM.Positie.Zoom";
      A(;
      L     "Positionering".Recept_Zoom;
      L     4;
      ==I;
      );
      JNB   _012;
      L     "Positionering".Recept4;
      T     DB4.DBB 0;
_012: NOP   0;
NETWORK
TITLE = Simualtie positionering
      A     "SIM.Positie.Zoom";
      A(;
      L     "Positionering".Recept_Zoom;
      L     5;
      ==I;
      );
      JNB   _013;
      L     "Positionering".Recept5;
      T     DB4.DBB 0;
_013: NOP   0;
NETWORK
TITLE = Simualtie positionering
      A     "SIM.Positie.Zoom";
      A(;
      L     "Positionering".Recept_Zoom;
      L     6;
      ==I;
      );
      JNB   _014;
      L     "Positionering".Recept6;
      T     DB4.DBB 0;
_014: NOP   0;
NETWORK
TITLE = Simualtie positionering
      A     "SIM.Positie.Zoom";
      A(;
      L     "Positionering".Recept_Zoom;
      L     7;
      ==I;
      );
      JNB   _015;
      L     "Positionering".Recept7;
      T     DB4.DBB 0;
_015: NOP   0;
NETWORK
TITLE = Simualtie positionering
      A     "SIM.Positie.Zoom";
      A(;
      L     "Positionering".Recept_Zoom;
      L     8;
      ==I;
      );
      JNB   _016;
      L     "Positionering".Recept8;
      T     DB4.DBB 0;
_016: NOP   0;
NETWORK
TITLE = Simualtie positionering
      A     "SIM.Positie.Zoom";
      A(;
      L     "Positionering".Recept_Zoom;
      L     9;
      ==I;
      );
      JNB   _017;
      L     "Positionering".Recept9;
      T     DB4.DBB 0;
_017: NOP   0;
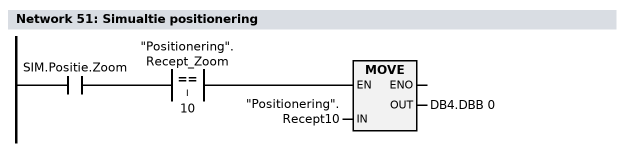
NETWORK
TITLE = Simualtie positionering
      A     "SIM.Positie.Zoom";
      A(;
      L     "Positionering".Recept_Zoom;
      L     10;
      ==I;
      );
      JNB   _018;
      L     "Positionering".Recept10;
      T     DB4.DBB 0;
_018: NOP   0;
END_FUNCTION

FUNCTION "Opstart_FC" : VOID	// FC 6
VERSION : 0.1
BEGIN
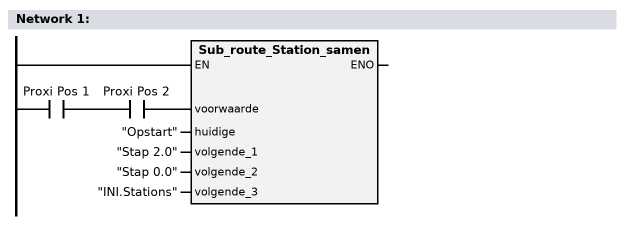
NETWORK
TITLE =
      A     "Proxi Pos 1";
      A     "Proxi Pos 2";
      =     L 0.0;
      BLD   103;
      CALL  "Sub_route_Station_samen" (
           voorwaarde               := L 0.0,
           huidige                  := "Opstart",
           volgende_1               := "Stap 2.0",
           volgende_2               := "Stap 0.0",
           volgende_3               := "INI.Stations");
      NOP   0;
END_FUNCTION

FUNCTION "Grafcet_Platform" : VOID	// FC 7
VERSION : 0.1
BEGIN
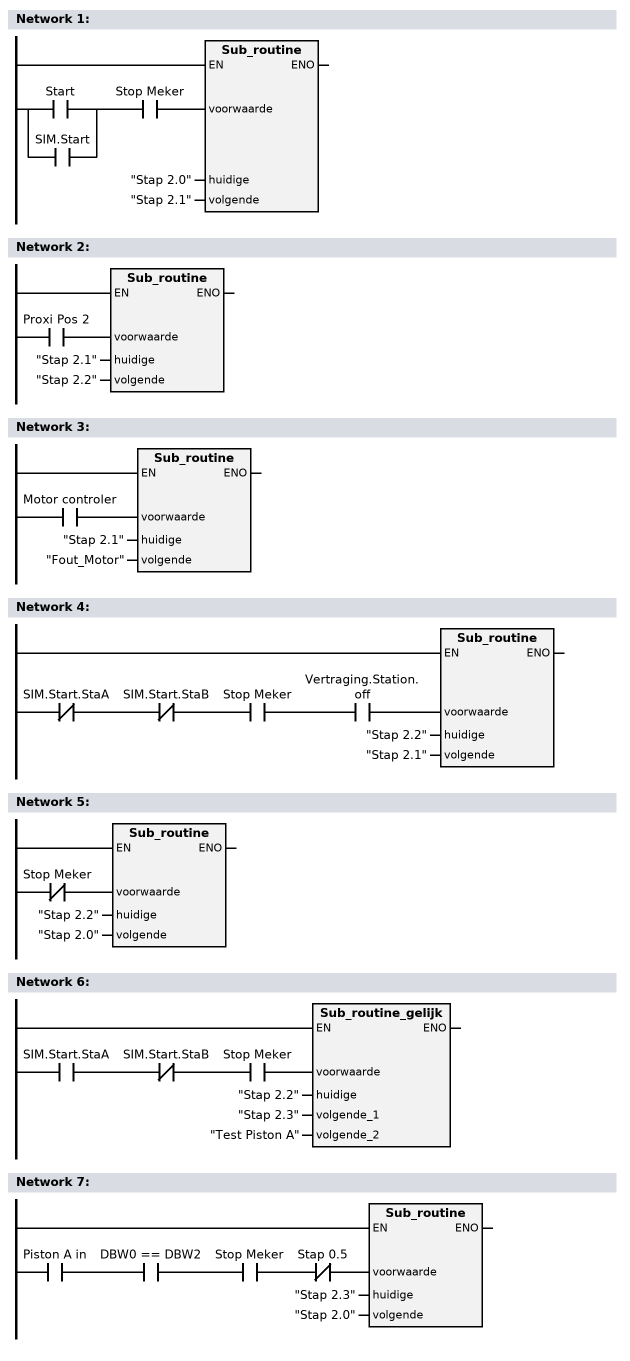
NETWORK
TITLE =
      A(;
      O     "Start";
      O     "SIM.Start";
      );
      A     "Stop Meker";
      =     L 0.0;
      BLD   103;
      CALL  "Sub_routine" (
           voorwaarde               := L 0.0,
           huidige                  := "Stap 2.0",
           volgende                 := "Stap 2.1");
      NOP   0;
NETWORK
TITLE =
      A     "Proxi Pos 2";
      =     L 0.0;
      BLD   103;
      CALL  "Sub_routine" (
           voorwaarde               := L 0.0,
           huidige                  := "Stap 2.1",
           volgende                 := "Stap 2.2");
      NOP   0;
NETWORK
TITLE =
      A     "Motor controler";
      =     L 0.0;
      BLD   103;
      CALL  "Sub_routine" (
           voorwaarde               := L 0.0,
           huidige                  := "Stap 2.1",
           volgende                 := "Fout_Motor");
      NOP   0;
NETWORK
TITLE =
      AN    "SIM.Start.StaA";
      AN    "SIM.Start.StaB";
      A     "Stop Meker";
      A     "Vertraging.Station.off";
      =     L 0.0;
      BLD   103;
      CALL  "Sub_routine" (
           voorwaarde               := L 0.0,
           huidige                  := "Stap 2.2",
           volgende                 := "Stap 2.1");
      NOP   0;
NETWORK
TITLE =
      AN    "Stop Meker";
      =     L 0.0;
      BLD   103;
      CALL  "Sub_routine" (
           voorwaarde               := L 0.0,
           huidige                  := "Stap 2.2",
           volgende                 := "Stap 2.0");
      NOP   0;
NETWORK
TITLE =
      A     "SIM.Start.StaA";
      AN    "SIM.Start.StaB";
      A     "Stop Meker";
      =     L 0.0;
      BLD   103;
      CALL  "Sub_routine_gelijk" (
           voorwaarde               := L 0.0,
           huidige                  := "Stap 2.2",
           volgende_1               := "Stap 2.3",
           volgende_2               := "Test Piston A");
      NOP   0;
NETWORK
TITLE =
      A     "Piston A in";
      A     "DBW0 == DBW2";
      A     "Stop Meker";
      AN    "Stap 0.5";
      =     L 0.0;
      BLD   103;
      CALL  "Sub_routine" (
           voorwaarde               := L 0.0,
           huidige                  := "Stap 2.3",
           volgende                 := "Stap 2.0");
      NOP   0;
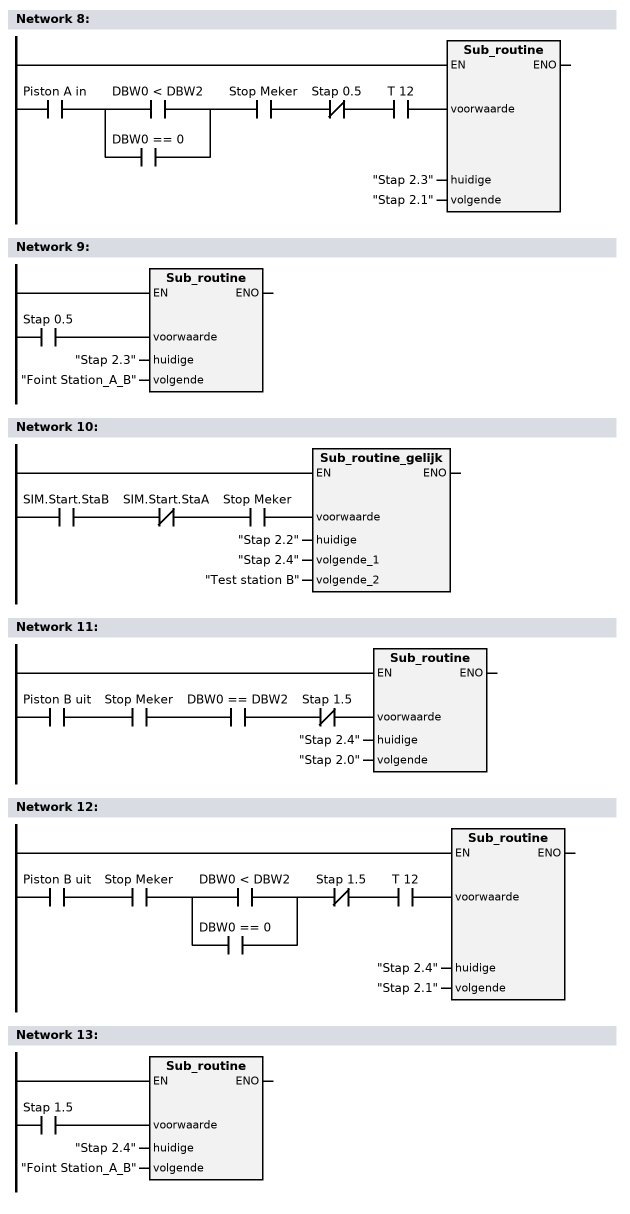
NETWORK
TITLE =
      A     "Piston A in";
      A(;
      O     "DBW0 < DBW2";
      O     "DBW0 == 0";
      );
      A     "Stop Meker";
      AN    "Stap 0.5";
      A     T 12;
      =     L 0.0;
      BLD   103;
      CALL  "Sub_routine" (
           voorwaarde               := L 0.0,
           huidige                  := "Stap 2.3",
           volgende                 := "Stap 2.1");
      NOP   0;
NETWORK
TITLE =
      A     "Stap 0.5";
      =     L 0.0;
      BLD   103;
      CALL  "Sub_routine" (
           voorwaarde               := L 0.0,
           huidige                  := "Stap 2.3",
           volgende                 := "Foint Station_A_B");
      NOP   0;
NETWORK
TITLE =
      A     "SIM.Start.StaB";
      AN    "SIM.Start.StaA";
      A     "Stop Meker";
      =     L 0.0;
      BLD   103;
      CALL  "Sub_routine_gelijk" (
           voorwaarde               := L 0.0,
           huidige                  := "Stap 2.2",
           volgende_1               := "Stap 2.4",
           volgende_2               := "Test station B");
      NOP   0;
NETWORK
TITLE =
      A     "Piston B uit";
      A     "Stop Meker";
      A     "DBW0 == DBW2";
      AN    "Stap 1.5";
      =     L 0.0;
      BLD   103;
      CALL  "Sub_routine" (
           voorwaarde               := L 0.0,
           huidige                  := "Stap 2.4",
           volgende                 := "Stap 2.0");
      NOP   0;
NETWORK
TITLE =
      A     "Piston B uit";
      A     "Stop Meker";
      A(;
      O     "DBW0 < DBW2";
      O     "DBW0 == 0";
      );
      AN    "Stap 1.5";
      A     T 12;
      =     L 0.0;
      BLD   103;
      CALL  "Sub_routine" (
           voorwaarde               := L 0.0,
           huidige                  := "Stap 2.4",
           volgende                 := "Stap 2.1");
      NOP   0;
NETWORK
TITLE =
      A     "Stap 1.5";
      =     L 0.0;
      BLD   103;
      CALL  "Sub_routine" (
           voorwaarde               := L 0.0,
           huidige                  := "Stap 2.4",
           volgende                 := "Foint Station_A_B");
      NOP   0;
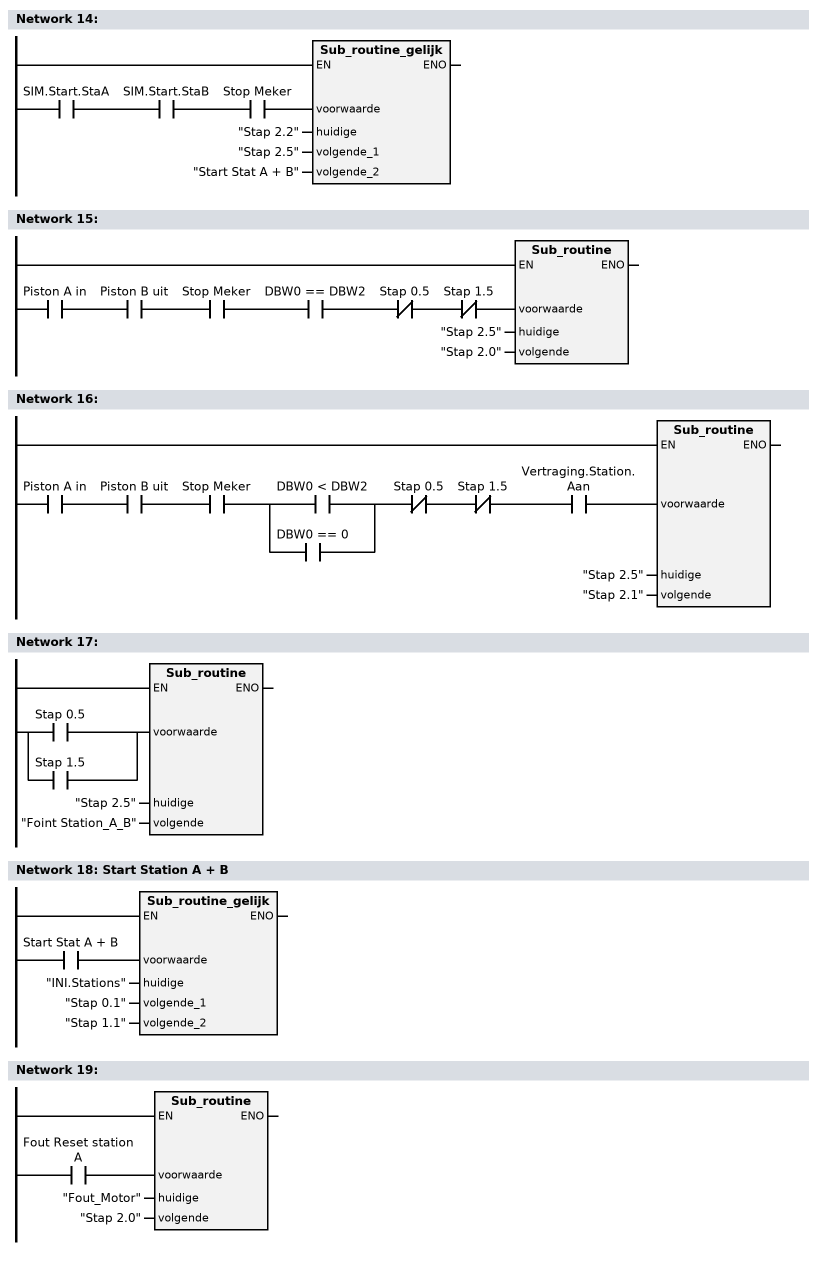
NETWORK
TITLE =
      A     "SIM.Start.StaA";
      A     "SIM.Start.StaB";
      A     "Stop Meker";
      =     L 0.0;
      BLD   103;
      CALL  "Sub_routine_gelijk" (
           voorwaarde               := L 0.0,
           huidige                  := "Stap 2.2",
           volgende_1               := "Stap 2.5",
           volgende_2               := "Start Stat A + B");
      NOP   0;
NETWORK
TITLE =
      A     "Piston A in";
      A     "Piston B uit";
      A     "Stop Meker";
      A     "DBW0 == DBW2";
      AN    "Stap 0.5";
      AN    "Stap 1.5";
      =     L 0.0;
      BLD   103;
      CALL  "Sub_routine" (
           voorwaarde               := L 0.0,
           huidige                  := "Stap 2.5",
           volgende                 := "Stap 2.0");
      NOP   0;
NETWORK
TITLE =
      A     "Piston A in";
      A     "Piston B uit";
      A     "Stop Meker";
      A(;
      O     "DBW0 < DBW2";
      O     "DBW0 == 0";
      );
      AN    "Stap 0.5";
      AN    "Stap 1.5";
      A     "Vertraging.Station.Aan";
      =     L 0.0;
      BLD   103;
      CALL  "Sub_routine" (
           voorwaarde               := L 0.0,
           huidige                  := "Stap 2.5",
           volgende                 := "Stap 2.1");
      NOP   0;
NETWORK
TITLE =
      A(;
      O     "Stap 0.5";
      O     "Stap 1.5";
      );
      =     L 0.0;
      BLD   103;
      CALL  "Sub_routine" (
           voorwaarde               := L 0.0,
           huidige                  := "Stap 2.5",
           volgende                 := "Foint Station_A_B");
      NOP   0;
NETWORK
TITLE = Start Station A + B
      A     "Start Stat A + B";
      =     L 0.0;
      BLD   103;
      CALL  "Sub_routine_gelijk" (
           voorwaarde               := L 0.0,
           huidige                  := "INI.Stations",
           volgende_1               := "Stap 0.1",
           volgende_2               := "Stap 1.1");
      NOP   0;
NETWORK
TITLE =
      A     "Fout Reset station A";
      =     L 0.0;
      BLD   103;
      CALL  "Sub_routine" (
           voorwaarde               := L 0.0,
           huidige                  := "Fout_Motor",
           volgende                 := "Stap 2.0");
      NOP   0;
END_FUNCTION

FUNCTION "Ingang -> Merker" : VOID	// FC 8
VERSION : 0.1
BEGIN
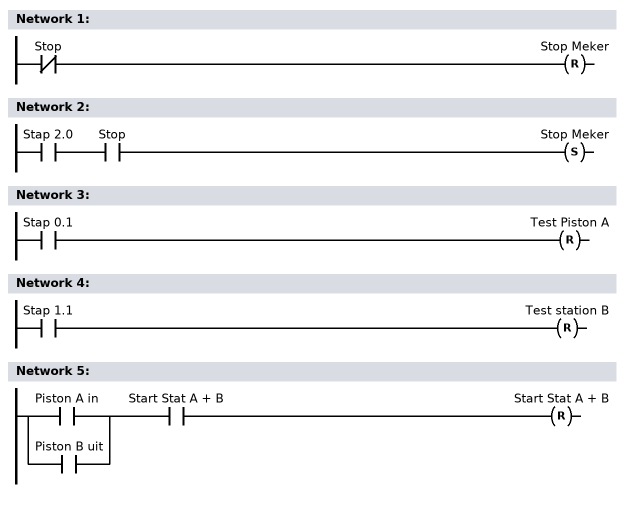
NETWORK
TITLE =
      AN    "Stop";
      R     "Stop Meker";
NETWORK
TITLE =
      A     "Stap 2.0";
      A     "Stop";
      S     "Stop Meker";
NETWORK
TITLE =
      A     "Stap 0.1";
      R     "Test Piston A";
NETWORK
TITLE =
      A     "Stap 1.1";
      R     "Test station B";
NETWORK
TITLE =
      A(;
      O     "Piston A in";
      O     "Piston B uit";
      );
      A     "Start Stat A + B";
      R     "Start Stat A + B";
END_FUNCTION

FUNCTION "DB_Function" : VOID	// FC 9
VERSION : 0.1
BEGIN
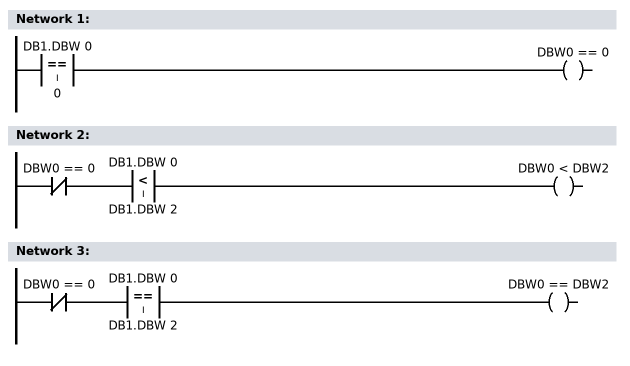
NETWORK
TITLE =
      L     DB1.DBW 0;
      L     0;
      ==I;
      =     "DBW0 == 0";
NETWORK
TITLE =
      AN    "DBW0 == 0";
      A(;
      L     DB1.DBW 0;
      L     DB1.DBW 2;
      <I;
      );
      =     "DBW0 < DBW2";
NETWORK
TITLE =
      AN    "DBW0 == 0";
      A(;
      L     DB1.DBW 0;
      L     DB1.DBW 2;
      ==I;
      );
      =     "DBW0 == DBW2";
END_FUNCTION

FUNCTION "SIM.OB100" : VOID	// FC 10
VERSION : 0.1
BEGIN
